Universal Robots URScript: move_path_cover_straight.script

def move_path_cover_straight():
  global _hidden_verificationVariable=0
  set_target_payload(10.800000, [-0.001000, -0.053000, 0.068000], [0.081228, 0.081228, 0.081228, 0.000000, 0.000000, 0.000000])
  set_gravity([0.0, 0.0, 9.82])
  set_standard_analog_input_domain(0, 1)
  set_standard_analog_input_domain(1, 1)
  set_tool_analog_input_domain(0, 1)
  set_tool_analog_input_domain(1, 1)
  set_analog_outputdomain(0, 0)
  set_analog_outputdomain(1, 0)
  set_input_actions_to_default()
  set_safety_mode_transition_hardness(1)
  set_tcp(p[-0.0095,-0.328,0.10573,1.2092,-1.2092,1.2092])
  set_tool_communication(False, 115200, 0, 1, 1.5, 3.5)
  set_tool_output_mode(0)
  set_tool_digital_output_mode(0, 1)
  set_tool_digital_output_mode(1, 1)
  set_tool_voltage(0)
  global robot_number=2
  global Point_1=p[0.0,0.0,0.0,0.0,0.0,0.0]
  global Point_2=p[0.0,0.0,0.0,0.0,0.0,0.0]
  # begin: URCap Installation Node
  #   Source: UR Connect, 1.13.79, Universal Robots
  #   Type: UR Connect
  myurRPC = rpc_factory("xmlrpc","http://127.0.0.1:40474")
  # end: URCap Installation Node
  # begin: URCap Installation Node
  #   Source: MachineLogic for Universal Robots, 3.1.7, Vention Inc.
  #   Type: MachineLogic for Universal Robots
  def waitForResponse(expected_response_vention, cname_vention):
  response_vention = socket_read_string(cname_vention,timeout=15)
  while response_vention != expected_response_vention:
  sleep(0.01)
  response_vention = socket_read_string(cname_vention,timeout=15)
  end
  sleep(0.01)
  sync()
  end
  def sendString(string_vention, expected_response_vention, cname_vention):
  socket_send_string(str_cat(string_vention,";"), cname_vention)
  response_vention = socket_read_string(cname_vention,timeout=15)
  if(response_vention == "nAck"):
  popup("nAck received")
  end
  while response_vention != expected_response_vention:
  sleep(0.01)
  response_vention = socket_read_string(cname_vention,timeout=15)
  if(response_vention == "nAck"):
  popup("nAck received")
  end
  end
  sleep(0.01)
  sync()
  end
  def sendStringNAck(string_vention, expected_response_vention, cname_vention):
  socket_send_string(str_cat(string_vention,";"), cname_vention)
  response_vention = socket_read_string(cname_vention,timeout=15)
  if(response_vention == "nAck"):
  popup("nAck received")
  end
  while(response_vention != expected_response_vention and response_vention != "nAck"):
  sleep(0.01)
  response_vention = socket_read_string(cname_vention,timeout=15)
  if(response_vention == "nAck"):
  popup("nAck received",blocking=True)
  end
  end
  sleep(0.01)
  sync()
  end
  def sendStringWithTimeout(string_vention, expected_response_vention, cname_vention):
  socket_send_string(str_cat(string_vention,";"), cname_vention)
  response_vention = socket_read_string(cname_vention,timeout=10)
  if(response_vention == "nAck"):
  popup("nAck received"+string_vention)
  end
  sleep(0.01)
  sync()
  end
  def pollString(string_vention, expected_response_vention, cname_vention):
  socket_send_string(str_cat(string_vention,";"), cname_vention)
  response_vention = socket_read_string(cname_vention,timeout=15)
  if(response_vention == "nAck"):
  popup("nAck received")
  end
  while response_vention != expected_response_vention:
  sleep(1)
  socket_send_string(str_cat(string_vention,";"), cname_vention)
  response_vention = socket_read_string(cname_vention,timeout=15)
  if(response_vention == "nAck"):
  popup("nAck received")
  end
  end
  sleep(0.01)
  sync()
  end
  def sendVariable(var_vention, data_vention, expected_response_vention, cname_vention):
  socket_set_var(var_vention, data_vention, cname_vention)
  response_vention = socket_read_string(cname_vention,timeout=15)
  if(response_vention == "nAck"):
  popup("nAck received")
  end
  while response_vention != expected_response_vention:
  sleep(0.01)
  response_vention = socket_read_string(cname_vention,timeout=15)
  if(response_vention == "nAck"):
  popup("nAck received")
  end
  end
  sleep(0.01)
  sync()
  end
  def intToString(integer_vention,cname_vention):
  stringFix=""
  multiplier_vention123=1
  if integer_vention<0:
  stringFix="-"
  multiplier_vention123=-1
  end
  socket_set_var("GetString",integer_vention*multiplier_vention123,cname_vention)
  string_vention=""
  while string_vention=="":
  sleep(0.01)
  string_vention=socket_read_string(cname_vention,timeout=15)
  end
  sleep(0.01)
  sync()
  string_vention=stringFix+string_vention
  return string_vention
  end
  string_vention=""
  isVentionMovementBusy = False
  isVentionParallelMovementSendingScript = False
  ventionThreadHandle = 1
  isVentionMovementBusyMachineMotion1 = False
  isVentionParallelMovementSendingScriptMachineMotion1 = False
  socket_vention = socket_open("192.168.3.52", 9999, "MachineMotion1")
  if socket_vention==False:
  popup("Check configuration, can't connect to MachineMotion")
  end
  waitForResponse("MachineMotion connection established", "MachineMotion1")
  sendString("isReady", "MachineMotion isReady = true", "MachineMotion1")
  sendStringWithTimeout("setURCapVersion2", "setURCapVersion loaded", "MachineMotion1")
  sendString("SET speed_v2 1000000", "Ack", "MachineMotion1")
  sendString("SET acceleration_v2 100000", "Ack", "MachineMotion1")
  sendString("SET de_axis_1_microsteps_config 8", "Ack", "MachineMotion1")
  sendString("SET de_axis_1_mechanical_gain_config_v2 150000.0", "Ack", "MachineMotion1")
  sendString("SET de_axis_1_direction_config 1", "Ack", "MachineMotion1")
  sendString("SET de_axis_1_type_config Custom Actuator ", "Ack", "MachineMotion1")
  sendString("de_axis_1_config_exec", "Ack", "MachineMotion1")
  # end: URCap Installation Node
  # begin: URCap Installation Node
  #   Source: WireTank Serial, 4.9.0, WireTank, LLC
  #   Type: WireTank Serial
  WTSerialBridge = rpc_factory("xmlrpc","http://127.0.0.1:40511/RPC2")
  # end: URCap Installation Node
  step_count_cfc27bff_3819_45be_bfcf_d52b1b1e9d2e = 0.0
  thread Step_Counter_Thread_60c3a4a9_e978_4eed_be39_a7f2d0dbddbc():
    while (True):
      step_count_cfc27bff_3819_45be_bfcf_d52b1b1e9d2e = step_count_cfc27bff_3819_45be_bfcf_d52b1b1e9d2e + 1.0
      sync()
    end
  end
  run Step_Counter_Thread_60c3a4a9_e978_4eed_be39_a7f2d0dbddbc()
  $ 2 "Robot Program"
  $ 3 "p1≔pathturn[1]"
  global p1=pathturn[1]
  $ 4 "p2≔pathturn[2]"
  global p2=pathturn[2]
  $ 5 "p3≔pathturn[3]"
  global p3=pathturn[3]
  $ 6 "p4≔pathturn[4]"
  global p4=pathturn[4]
  $ 7 "p5≔pathturn[5]"
  global p5=pathturn[5]
  $ 8 "p6≔pathturn[6]"
  global p6=pathturn[6]
  $ 9 "pa1≔p[p1[0],p1[1],p1[2]+0.05,p1[3],p1[4],p1[5]]"
  global pa1=p[p1[0],p1[1],p1[2]+0.05,p1[3],p1[4],p1[5]]
  $ 10 "pret≔p[p6[0],p6[1],p6[2]+0.05,p6[3],p6[4],p6[5]]"
  global pret=p[p6[0],p6[1],p6[2]+0.05,p6[3],p6[4],p6[5]]
  $ 11 "'go to preheat'"
  # 'go to preheat'
  $ 12 "Set"
  set_tcp(p[-0.0095,-0.328,0.10573,1.2092,-1.2092,1.2092])
  $ 13 "MoveJ"
  $ 14 "pa1" "breakAfter"
  movej(pa1, a=1.3962634015954636, v=1.0471975511965976)
  $ 15 "MoveL"
  $ 16 "p1" "breakAfter"
  movel(p1, a=0.05, v=0.05)
  $ 17 "Wait: 4.0"
  sleep(4.0)
  # begin: URCap Program Node
  #   Source: WireTank Serial, 4.9.0, WireTank, LLC
  #   Type: WireTank Serial
  $ 18 "Serial Bridge uR1"
  SerialResponse = WTSerialBridge.send_command("/dev/ttyUSB0",1200, 8, "None", "One", "None", 1000, "None", "None", [252,82,49], False)
  # end: URCap Program Node
  $ 19 "Set DO[0]=On"
  set_standard_digital_out(0, True)
  $ 20 "Wait: 1.0"
  sleep(1.0)
  $ 21 "MoveL"
  $ 22 "p2" "breakAfter"
  movel(p2, a=1.2, v=0.01)
  $ 23 "p3" "breakAfter"
  movel(p3, a=1.2, v=0.01)
  $ 24 "p4" "breakAfter"
  movel(p4, a=1.2, v=0.01)
  $ 25 "p5" "breakAfter"
  movel(p5, a=1.2, v=0.01)
  # begin: URCap Program Node
  #   Source: WireTank Serial, 4.9.0, WireTank, LLC
  #   Type: WireTank Serial
  $ 26 "Serial Bridge uR0"
  SerialResponse = WTSerialBridge.send_command("/dev/ttyUSB0",1200, 8, "None", "One", "None", 1000, "None", "None", [252,82,48], False)
  # end: URCap Program Node
  $ 27 "Set DO[0]=Off"
  set_standard_digital_out(0, False)
  $ 28 "MoveL"
  $ 29 "p6" "breakAfter"
  movel(p6, a=1.2, v=0.01)
  $ 30 "Wait: 1.0"
  sleep(1.0)
  $ 31 "MoveL"
  $ 32 "pret" "breakAfter"
  movel(pret, a=0.05, v=0.05)
end
